// TwinCAT 3 PLC project AdventOfCode2024_Day01
// ProgramVersion: 3.1.4026.12
// libraries:
//   Tc2_Standard, * (Beckhoff Automation GmbH)
//   Tc2_System, * (Beckhoff Automation GmbH)
//   Tc2_Utilities, * (Beckhoff Automation GmbH)
// project tree:
//   DUTs/ ERROR.TcDUT
//   GVLs/ GLOBAL_CONSTANTS.TcGVL
//   / PlcTask.TcTTO
//   POUs/ BubbleSort.TcPOU, MAIN.TcPOU
//   POUs/FileReader/DUTs/ STATE.TcDUT
//   POUs/FileReader/ FileReader.TcPOU
// real-time tasks:
//   TASK PlcTask: cycle T#10ms, priority 20, ADS port 350

CONFIGURATION AdventOfCode2024_Day01
    RESOURCE PLC ON TwinCAT3
        TASK PlcTask(INTERVAL := T#10ms, PRIORITY := 20);
        PROGRAM MAIN WITH PlcTask : MAIN;
    END_RESOURCE
END_CONFIGURATION

// ---- DUTs/ERROR.TcDUT
TYPE ERROR :
STRUCT
	bError : BOOL;
	nErrorCode : UDINT;
	dtCurrentTime : DT;
END_STRUCT
END_TYPE

// ---- POUs/FileReader/DUTs/STATE.TcDUT
{attribute 'qualified_only'}
{attribute 'strict'}
{attribute 'to_string'}
TYPE STATE :
(
	Idle := 0,
	OpenFile := 1,
	OpenFileAwaitFinish := 2,
	ReadFile := 3,
	ReadFileAwaitFinish := 4,
	CloseFile := 5,
	CloseFileAwaitFinish := 6,
	Error := 99
);
END_TYPE

// ---- GVLs/GLOBAL_CONSTANTS.TcGVL
VAR_GLOBAL CONSTANT
	iC_MAX_NUM_LINES_IN_FILE : UINT := 999;
	iC_MAX_STRING_LENGTH : UINT := 50;
END_VAR

// ---- POUs/MAIN.TcPOU
PROGRAM MAIN
VAR
	fbSystemTime : GETSYSTEMTIME;
    timeAsFileTime : T_FILETIME;
    timeAsDT : DT;	

	fbi_FileReader : FileReader;
	
	sFilePath : T_MaxString := 'E:\Projects\Twincat\AdventOfCode\Day01\Day1Input.txt'; //'C:\temp\HelloWorld.txt';// 
	
	arsFileContent : ARRAY [0..iC_MAX_NUM_LINES_IN_FILE] OF STRING(iC_MAX_STRING_LENGTH);
	ariFileContentA : ARRAY[0..iC_MAX_NUM_LINES_IN_FILE] OF UDINT;
	ariFileContentB : ARRAY[0..iC_MAX_NUM_LINES_IN_FILE] OF UDINT;
	iLoopIndexFileContentArray : UINT;
	jLoopIndexFileContentArray : UINT;
	sTempString : STRING;
	sTempStringSplit : STRING;
	sTempStringSplit2 : STRING;
	iDifference : DINT;
	
	iSumOfDifferences : DINT;
	iSumOfScore : DINT;
	
	bReadFile : BOOL;
	bConvertArray : BOOL;
	bCalcSimilarity2 : BOOL;
END_VAR

fbSystemTime(timeLoDW=>timeAsFileTime.dwLowDateTime, timeHiDW=>timeAsFileTime.dwHighDateTime);

fbi_FileReader();

IF bReadFile THEN
	bReadFile := FALSE;
	fbi_FileReader.ReadFile(sFilePath);
END_IF

IF bConvertArray THEN
	bConvertArray := FALSE;
	iLoopIndexFileContentArray := 0;
	iSumOfDifferences := 0;
	FOR iLoopIndexFileContentArray := 0 TO iC_MAX_NUM_LINES_IN_FILE DO
		sTempString := fbi_FileReader.GetLineByIndex(iLoopIndexFileContentArray);
		sTempStringSplit := MID(sTempString,5,1);
		sTempStringSplit2 := MID(sTempString,5,9);
		
		ariFileContentA[iLoopIndexFileContentArray] := TO_UDINT(sTempStringSplit);
		ariFileContentB[iLoopIndexFileContentArray] := TO_UDINT(sTempStringSplit2);													
	END_FOR
	BubbleSort(ariFileContentA);
	BubbleSort(ariFileContentB);
	FOR iLoopIndexFileContentArray := 0 TO iC_MAX_NUM_LINES_IN_FILE DO
		iDifference := ariFileContentA[iLoopIndexFileContentArray] - ariFileContentB[iLoopIndexFileContentArray];
				IF iDifference >= 0 THEN
					iSumOfDifferences := iSumOfDifferences + iDifference;
				ELSE
					iSumOfDifferences := iSumOfDifferences - iDifference; 	
				END_IF
	END_FOR	
END_IF

IF bCalcSimilarity2 THEN
	bCalcSimilarity2 := FALSE;
	iSumOfScore := 0;
	FOR iLoopIndexFileContentArray := 0 TO iC_MAX_NUM_LINES_IN_FILE DO
		FOR jLoopIndexFileContentArray := 0 TO iC_MAX_NUM_LINES_IN_FILE DO
			IF ariFileContentA[iLoopIndexFileContentArray] = ariFileContentB[jLoopIndexFileContentArray] THEN
				iSumOfScore := iSumOfScore + TO_DINT(ariFileContentA[iLoopIndexFileContentArray]);
			END_IF
		END_FOR
	END_FOR
END_IF

END_PROGRAM

// ---- POUs/FileReader/FileReader.TcPOU
FUNCTION_BLOCK FileReader
VAR
	_bBusy : BOOL;
	_sFilePath : STRING;
	_arsFileContent : ARRAY [0..iC_MAX_NUM_LINES_IN_FILE] OF STRING(iC_MAX_STRING_LENGTH);
	
	fbi_FileOpen : FB_FileOpen;
	fbi_FileGets : FB_FileGets;
	fbi_FileClose : FB_FileClose;
	
	eState : STATE := STATE.Idle;
	
	hFileHandle : UINT;
	iFileContentNextIndex : UINT;
	stError : ERROR;
END_VAR

CASE eState OF
	State.Idle:
		// Do nothing
	State.OpenFile:
		_bBusy := TRUE;
		iFileContentNextIndex := 0;
		MEMSET(ADR(_arsFileContent), 0, SIZEOF(_arsFileContent));
		fbi_FileOpen(sPathName := sFilePath, nMode := FOPEN_MODEREAD OR FOPEN_MODETEXT, ePath := PATH_GENERIC, bExecute := TRUE, bError => stError.bError, nErrId => stError.nErrorCode);
		eState := STATE.OpenFileAwaitFinish;
		
	State.OpenFileAwaitFinish:
		fbi_FileOpen(bExecute := FALSE, hFile => hFileHandle, bError => stError.bError, nErrId => stError.nErrorCode);
		IF NOT fbi_FileOpen.bBusy THEN
			IF NOT stError.bError THEN
				eState := STATE.ReadFile;
			ELSE
				eState := STATE.Error;
			END_IF
		END_IF
		
	State.ReadFile:
		fbi_FileGets(hFile := hFileHandle, bExecute := TRUE, bError => stError.bError, nErrId => stError.nErrorCode);
		eState := STATE.ReadFileAwaitFinish;
		
	State.ReadFileAwaitFinish:
		fbi_FileGets(bExecute := FALSE, bError => stError.bError, nErrId => stError.nErrorCode);
		IF NOT fbi_FileGets.bBusy THEN
			IF NOT stError.bError THEN
				_arsFileContent[iFileContentNextIndex] := fbi_FileGets.sLine;
				IF fbi_FileGets.bEOF THEN
					eState := STATE.CloseFile;
				ELSE
					eState := STATE.ReadFile;
					iFileContentNextIndex := iFileContentNextIndex+1;	
				END_IF
			ELSE
				eState := STATE.Error;
			END_IF	
		END_IF
		
	State.CloseFile:
		fbi_FileClose(hFile := hFileHandle, bExecute := TRUE, bError => stError.bError, nErrId => stError.nErrorCode);
		eState := STATE.CloseFileAwaitFinish;
		
	State.CloseFileAwaitFinish:
		fbi_FileClose(bExecute := FALSE, bError => stError.bError, nErrId => stError.nErrorCode);
		IF NOT fbi_FileClose.bBusy THEN
			IF NOT stError.bError THEN
				eState := STATE.Idle;
			ELSE
				eState := STATE.Error;
			END_IF
			_bBusy := FALSE;
			hFileHandle := 0;
		END_IF
		
	State.Error:
		stError.dtCurrentTime := FILETIME_TO_DT(MAIN.timeAsFileTime);
		eState := STATE.Idle;
END_CASE

PROPERTY arsFileContent : ARRAY [0..iC_MAX_NUM_LINES_IN_FILE] OF STRING(iC_MAX_STRING_LENGTH)
GET
arsFileContent := _arsFileContent;
END_GET
END_PROPERTY

PROPERTY bBusy : BOOL
GET
bBusy := _bBusy;
END_GET
END_PROPERTY

METHOD GetLineByIndex : STRING
VAR_INPUT
	iIndex : UINT;
END_VAR
GetLineByIndex := _arsFileContent[iIndex];
END_METHOD

METHOD ReadFile : BOOL
VAR_INPUT
	sFilePath : STRING;
END_VAR
_bBusy := TRUE;
_sFilePath := sFilePath;
IF eState = STATE.Idle THEN
	eState := STATE.OpenFile;
END_IF
ReadFile := NOT _bBusy AND NOT stError.bError;
END_METHOD

PROPERTY sFilePath : STRING
GET
sFilePath := _sFilePath;
END_GET
SET
_sFilePath := sFilePath;
END_SET
END_PROPERTY

END_FUNCTION_BLOCK

// ---- POUs/BubbleSort.TcPOU
FUNCTION BubbleSort : BOOL
VAR_IN_OUT
	arrValues : ARRAY[0..iC_MAX_NUM_LINES_IN_FILE] OF UDINT;
END_VAR
VAR
	i, j : UDINT;
	temp : UDINT;
END_VAR

// Bubble Sort Algorithmus
FOR i := 0 TO iC_MAX_NUM_LINES_IN_FILE-1 DO
    FOR j := 0 TO iC_MAX_NUM_LINES_IN_FILE-1 DO
        IF arrValues[j] > arrValues[j + 1] THEN
            // Werte tauschen
            temp := arrValues[j];
            arrValues[j] := arrValues[j + 1];
            arrValues[j + 1] := temp;
        END_IF
    END_FOR
END_FOR;

END_FUNCTION
